// TIA Portal project "demo" (V15.1)

(* hardware
DEVICE "S7-1200 station_1"  S7-1200 Station
   slot 0: "Rack_0"  S7-1200 Rack  Rack  V1.0
   slot 1: "PLC_1"  CPU 1211C DC/DC/DC  6ES7 211-1AE40-0XB0  V4.2
*)

// ===== PLC "PLC_1"  CPU 1211C DC/DC/DC =====

VAR_GLOBAL   // PLC tag table "Default tag table"
   "Start" AT %I0.1 : Bool;
   "M_Start" AT %M0.0 : Bool;
   "Stop" AT %I0.3 : Bool;
   "Emergency stop" AT %I0.4 : Bool;
   "Reset" AT %I0.2 : Bool;
   "M_stop" AT %M0.1 : Bool;
   "M_reset" AT %M0.2 : Bool;
   "M_processing" AT %M0.3 : Bool;
   "Manual" AT %I0.6 : Bool;
   "Auto" AT %I0.5 : Bool;
   "Stop entry conveyor" AT %M0.4 : Bool;
   "Entry conveyor" AT %Q0.0 : Bool;
   "Exit conveyor" AT %Q0.2 : Bool;
   "Vision sensor" AT %ID30 : DInt;
   "M_vison_sensor" AT %M0.5 : Bool;
   "At exit" AT %I0.0 : Bool;
   "Sorter 1 belt" AT %Q0.4 : Bool;
   "Sorter 1 turn" AT %Q0.3 : Bool;
   "Sorter 2 belt" AT %Q0.6 : Bool;
   "Sorter 2 turn" AT %Q0.5 : Bool;
   "Sorter 3 belt" AT %Q1.0 : Bool;
   "Sorter 3 turn" AT %Q0.7 : Bool;
   "Counter 1" AT %QD30 : DInt;
   "Counter 2" AT %QD34 : DInt;
   "Counter 3" AT %QD38 : DInt;
   "Reset light" AT %Q1.2 : Bool;
   "Stop Light" AT %Q1.3 : Bool;
   "Start Light" AT %Q1.1 : Bool;
END_VAR

// folder: System blocks/Program resources

DATA_BLOCK "TON_1s"   // DB1
{ S7_Optimized_Access := 'TRUE' }
AUTHOR : Simatic
FAMILY : IEC
NAME : IEC_TMR
VERSION : 1.0
// stored: InstanceOfName IEC_TIMER
"IEC_TIMER"
BEGIN
END_DATA_BLOCK

DATA_BLOCK "CU1"   // DB2
{ S7_Optimized_Access := 'TRUE' }
AUTHOR : Simatic
FAMILY : IEC
NAME : CNTR
VERSION : 1.0
// stored: InstanceOfName IEC_COUNTER
"IEC_COUNTER"
BEGIN
END_DATA_BLOCK

DATA_BLOCK "CU2"   // DB3
{ S7_Optimized_Access := 'TRUE' }
AUTHOR : Simatic
FAMILY : IEC
NAME : CNTR
VERSION : 1.0
// stored: InstanceOfName IEC_COUNTER
"IEC_COUNTER"
BEGIN
END_DATA_BLOCK

DATA_BLOCK "CU3"   // DB4
{ S7_Optimized_Access := 'TRUE' }
AUTHOR : Simatic
FAMILY : IEC
NAME : CNTR
VERSION : 1.0
// stored: InstanceOfName IEC_COUNTER
"IEC_COUNTER"
BEGIN
END_DATA_BLOCK

// folder: (top level)

FUNCTION "MHJ-PLC-Lab-Function-S71200" : Void   // FC9000, SCL
{ S7_Optimized_Access := 'TRUE' }
VERSION : 0.1
   VAR_TEMP
      rdTimeReturn : Int;
      outputTime : DTL;
      SyncVal : Byte;
      forVal : Int;
      forVal_2 : Int;
      Value : Byte;
   END_VAR
   VAR CONSTANT
      CompVal : Byte := 16#34;
      Value_01 : Byte := 16#11;
      Value_01_DW : DWord := 16#A165_D992;
      Value_02_DW : DWord := 16#58BE_4401;
   END_VAR
BEGIN

   #Value:=PEEK(area := 16#82,
        dbNumber := 0,
        byteOffset := 511);
   #Value := #Value + 1;

   POKE(area := 16#82,
        dbNumber := 0,
        byteOffset := 511,
        value := #Value);

   POKE(area:=16#81,
        dbNumber:=0,
        byteOffset:=1016,
        value:=#Value_01_DW);
   POKE(area := 16#81,
        dbNumber := 0,
        byteOffset := 1020,
        value := #Value_02_DW);

   POKE(area := 16#81,
        dbNumber := 0,
        byteOffset := 511,
        value := B#16#00);

   FOR #forVal := 0 TO 120 DO
       FOR #forVal_2:=0 TO 10 DO
           #rdTimeReturn:=RD_SYS_T(#outputTime);
           #rdTimeReturn := WR_SYS_T(#outputTime);
           #rdTimeReturn := RD_SYS_T(#outputTime);
           #rdTimeReturn := WR_SYS_T(#outputTime);
       END_FOR;
       #SyncVal:= PEEK(area := 16#81,
                      dbNumber := 0,
                      byteOffset := 511);
       IF #SyncVal = #CompVal THEN
          GOTO M_1;
       END_IF;
   END_FOR;
   RETURN;

   M_1:
   POKE(area := 16#81,
        dbNumber := 0,
        byteOffset := 511,
        value := B#16#0);
END_FUNCTION

ORGANIZATION_BLOCK "Main"   // OB1, LAD, ProgramCycle
TITLE = "Main Program Sweep (Cycle)"
{ S7_Optimized_Access := 'TRUE' }
VERSION : 0.1
   VAR_INPUT
      Initial_Call : Bool;   // Initial call of this OB
      Remanence : Bool;   // =True, if remanent data are available
   END_VAR
BEGIN

REGION Network 1
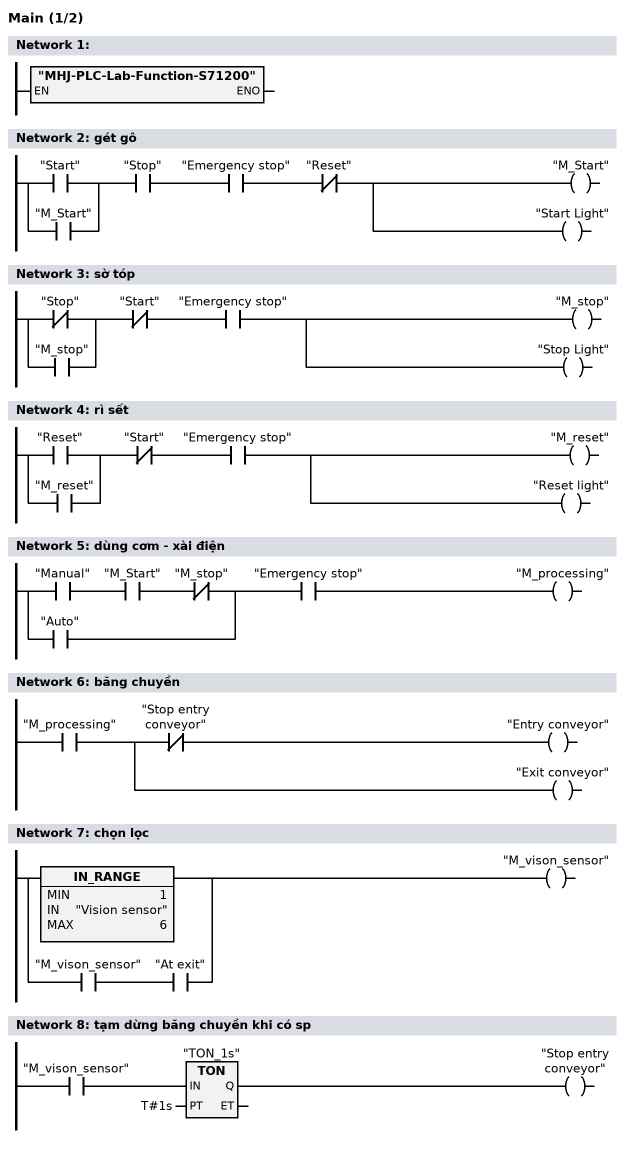
   RUNG wire#powerrail
      "MHJ-PLC-Lab-Function-S71200"()
   END_RUNG
   // the same network as SCL:
   "MHJ-PLC-Lab-Function-S71200"();
END_REGION

REGION Network 2: gét gô
   RUNG wire#powerrail
      Contact( "Start" )
      wire#w1
      Contact( "Stop" )
      Contact( "Emergency stop" )
      I_Contact( "Reset" )
      wire#w2
      Coil( "M_Start" )
   END_RUNG
   RUNG wire#powerrail
      Contact( "M_Start" )
   END_RUNG wire#w1
   RUNG wire#w2
      Coil( "Start Light" )
   END_RUNG
   // the same network as SCL:
   "M_Start" := ("Start" OR "M_Start") AND "Stop" AND "Emergency stop" AND NOT "Reset";
   "Start Light" := "M_Start";
END_REGION

REGION Network 3: sờ tóp
   RUNG wire#powerrail
      I_Contact( "Stop" )
      wire#w1
      I_Contact( "Start" )
      Contact( "Emergency stop" )
      wire#w2
      Coil( "M_stop" )
   END_RUNG
   RUNG wire#powerrail
      Contact( "M_stop" )
   END_RUNG wire#w1
   RUNG wire#w2
      Coil( "Stop Light" )
   END_RUNG
   // the same network as SCL:
   "M_stop" := (NOT "Stop" OR "M_stop") AND NOT "Start" AND "Emergency stop";
   "Stop Light" := "M_stop";
END_REGION

REGION Network 4: rì sết
   RUNG wire#powerrail
      Contact( "Reset" )
      wire#w1
      I_Contact( "Start" )
      Contact( "Emergency stop" )
      wire#w2
      Coil( "M_reset" )
   END_RUNG
   RUNG wire#powerrail
      Contact( "M_reset" )
   END_RUNG wire#w1
   RUNG wire#w2
      Coil( "Reset light" )
   END_RUNG
   // the same network as SCL:
   "M_reset" := ("Reset" OR "M_reset") AND NOT "Start" AND "Emergency stop";
   "Reset light" := "M_reset";
END_REGION

REGION Network 5: dùng cơm - xài điện
   RUNG wire#powerrail
      Contact( "Manual" )
      Contact( "M_Start" )
      I_Contact( "M_stop" )
      wire#w1
      Contact( "Emergency stop" )
      Coil( "M_processing" )
   END_RUNG
   RUNG wire#powerrail
      Contact( "Auto" )
   END_RUNG wire#w1
   // the same network as SCL:
   "M_processing" := (("Manual" AND "M_Start" AND NOT "M_stop") OR "Auto") AND "Emergency stop";
END_REGION

REGION Network 6: băng chuyền
   RUNG wire#powerrail
      Contact( "M_processing" )
      wire#w1
      I_Contact( "Stop entry conveyor" )
      Coil( "Entry conveyor" )
   END_RUNG
   RUNG wire#w1
      Coil( "Exit conveyor" )
   END_RUNG
   // the same network as SCL:
   "Entry conveyor" := "M_processing" AND NOT "Stop entry conveyor";
   "Exit conveyor" := "M_processing";
END_REGION

REGION Network 7: chọn lọc
   RUNG wire#powerrail
      { S7_Templates := "SrcType := DInt" } InRange(min := 1, in := "Vision sensor", max := 6)
      wire#w1
      Coil( "M_vison_sensor" )
   END_RUNG
   RUNG wire#powerrail
      Contact( "M_vison_sensor" )
      Contact( "At exit" )
   END_RUNG wire#w1
   // the same network as SCL:
   "M_vison_sensor" := ((1 <= "Vision sensor") AND ("Vision sensor" <= 6)) OR ("M_vison_sensor" AND "At exit");
END_REGION

REGION Network 8: tạm dừng băng chuyền khi có sp
   "TON_1s".TON(IN := "M_vison_sensor", PT := T#1s);
   "Stop entry conveyor" := "TON_1s".Q;
END_REGION

REGION Network 9: xử lý phân lạo 1
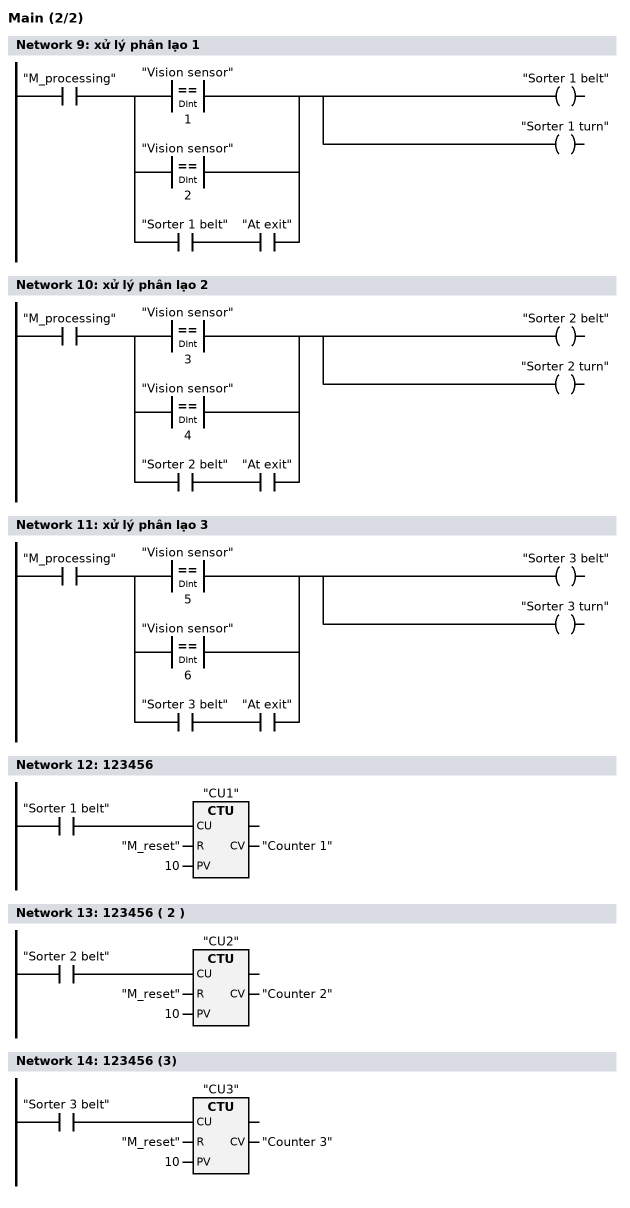
   RUNG wire#powerrail
      Contact( "M_processing" )
      wire#w1
      { S7_Templates := "SrcType := DInt" } EQ_Contact(in1 := "Vision sensor", in2 := 1)
      wire#w2
      Coil( "Sorter 1 belt" )
   END_RUNG
   RUNG wire#w1
      { S7_Templates := "SrcType := DInt" } EQ_Contact(in1 := "Vision sensor", in2 := 2)
   END_RUNG wire#w2
   RUNG wire#w1
      Contact( "Sorter 1 belt" )
      Contact( "At exit" )
   END_RUNG wire#w2
   RUNG wire#w2
      Coil( "Sorter 1 turn" )
   END_RUNG
   // the same network as SCL:
   "Sorter 1 belt" := "M_processing" AND (("Vision sensor" = 1) OR ("Vision sensor" = 2) OR ("Sorter 1 belt" AND "At exit"));
   "Sorter 1 turn" := "Sorter 1 belt";
END_REGION

REGION Network 10: xử lý phân lạo 2
   RUNG wire#powerrail
      Contact( "M_processing" )
      wire#w1
      { S7_Templates := "SrcType := DInt" } EQ_Contact(in1 := "Vision sensor", in2 := 3)
      wire#w2
      Coil( "Sorter 2 belt" )
   END_RUNG
   RUNG wire#w1
      { S7_Templates := "SrcType := DInt" } EQ_Contact(in1 := "Vision sensor", in2 := 4)
   END_RUNG wire#w2
   RUNG wire#w1
      Contact( "Sorter 2 belt" )
      Contact( "At exit" )
   END_RUNG wire#w2
   RUNG wire#w2
      Coil( "Sorter 2 turn" )
   END_RUNG
   // the same network as SCL:
   "Sorter 2 belt" := "M_processing" AND (("Vision sensor" = 3) OR ("Vision sensor" = 4) OR ("Sorter 2 belt" AND "At exit"));
   "Sorter 2 turn" := "Sorter 2 belt";
END_REGION

REGION Network 11: xử lý phân lạo 3
   RUNG wire#powerrail
      Contact( "M_processing" )
      wire#w1
      { S7_Templates := "SrcType := DInt" } EQ_Contact(in1 := "Vision sensor", in2 := 5)
      wire#w2
      Coil( "Sorter 3 belt" )
   END_RUNG
   RUNG wire#w1
      { S7_Templates := "SrcType := DInt" } EQ_Contact(in1 := "Vision sensor", in2 := 6)
   END_RUNG wire#w2
   RUNG wire#w1
      Contact( "Sorter 3 belt" )
      Contact( "At exit" )
   END_RUNG wire#w2
   RUNG wire#w2
      Coil( "Sorter 3 turn" )
   END_RUNG
   // the same network as SCL:
   "Sorter 3 belt" := "M_processing" AND (("Vision sensor" = 5) OR ("Vision sensor" = 6) OR ("Sorter 3 belt" AND "At exit"));
   "Sorter 3 turn" := "Sorter 3 belt";
END_REGION

REGION Network 12: 123456
   "CU1".CTU(CU := "Sorter 1 belt", R := "M_reset", PV := 10, CV => "Counter 1");
END_REGION

REGION Network 13: 123456 ( 2 )
   "CU2".CTU(CU := "Sorter 2 belt", R := "M_reset", PV := 10, CV => "Counter 2");
END_REGION

REGION Network 14: 123456 (3)
   "CU3".CTU(CU := "Sorter 3 belt", R := "M_reset", PV := 10, CV => "Counter 3");
END_REGION
END_ORGANIZATION_BLOCK